TYPE T_ProtobufRawBuffer : ARRAY[0..Param_PB.cMaxProtobufRawBuffer] OF BYTE; END_TYPE

(* stored: Version 1.1.0.1
   DUT T_ProtobufRawBuffer: Id {7dd154eb-fee9-4a02-a774-75ce0c6f4cd2} *)
